{attribute 'qualified_only'}
{attribute 'strict'}
{attribute 'to_string'}
TYPE SysteemStatusMogelijkheiden :
(
	Uit,
	Joggen,
	Locatie,
	Torque,
	PowerOff
);
END_TYPE

(* stored: Version 1.1.0.1, ProductVersion 3.1.4024.12
   EnumerationTextList DUT: Id {d2cd0a0b-263c-47b9-ba33-54791d0d5494} *)
